// TIA Portal V19 export
DATA_BLOCK "A0302_Bordatrice_PERS"   // DB44
// stored: MemoryReserve 100
   VAR RETAIN
      Par : Struct
         Ax_Man : "Positioning_EPOS_Machine_Par";
         Ax_Aut : "A0301_Mach_Speed_Par";
      END_STRUCT;
      Pers_Data : Struct
         EncoderAbsolute_Preset_OK : Bool := TRUE;
         Persistent_ActualPosition : LReal := 457025.036;
      END_STRUCT;
   END_VAR
BEGIN
   Par.Ax_Man.PosTolerance := 1.0;
   Par.Ax_Man.DelayInPosition := T#10MS;
   Par.Ax_Man.Man_Vel := 30000.0;
   Par.Ax_Man.Man_Acc := 1000.0;
   Par.Ax_Man.Man_Dec := 1000.0;
   Par.Ax_Aut.SemiAut_Vel := 40000.0;
   Par.Ax_Aut.Aut_Vel := 48000.0;
   Par.Ax_Aut.Aut_Acc := 1000.0;
   Par.Ax_Aut.Aut_Dec := 1000.0;
END_DATA_BLOCK
